Staubli VAL3: Input.pgx

program Input(num io, bool& value)
begin
  //*******************************************************************************
  //*   ______
  //*  / _____) /|
  //* | |      / /
  //* | | /\  / /
  //* | | \ \/ /  _      Copyright (c) KEOLABS, 2016
  //* | |  \__/  | |        http://www.keolabs.com
  //* | |________| |
  //*  \__________/
  //*
  //********************************************************************************
  //*@file          : Input
  //*@author        : Yves Ragot
  //*@version       : $Id: Input.pgx 1202 2016-10-07 12:12:19Z yves $
  //*@brief         : get Input value
  //*
  //*******************************************************************************/

   switch (io)

    case 1
        value = diVacuum
    break

    case 2
        value = difIn1
    break

    case 3
        value = diusrIn0
    break

    case 4
        value = diusrIn1
    break

    default
        GeneralStatus = 101
        LastErrorCode = 0
    break

  endSwitch

end
